{attribute 'analysis' := '-33'}
TYPE RbtFanucUnloading_GO :
STRUCT
	//GO[1]
	ErrorNr:UINT;
	State:UINT;
	NrPickedCrates:UINT;
	NrPayload:uint;
END_STRUCT
END_TYPE

(* stored: Version 1.1.0.1
   DUT RbtFanucUnloading_GO: Id {715d883e-3319-4687-b9af-8691602e5624} *)
